TYPE MultipleEventTestsystem :
STRUCT
  logging: EventRunner;
  event1: Event := (logging:=logging);
  event2: Event := (logging:=logging);
  event3: Event := (logging:=logging);
END_STRUCT
END_TYPE

(* stored: Version 1.1.0.1, ProductVersion 3.1.4024.9
   DUT MultipleEventTestsystem: Id {463db442-f089-4be4-9631-f04acbc95b47} *)
